FUNCTION_BLOCK T_MockStateModule IMPLEMENTS I_StateModule
VAR_INPUT
  _currentState : UINT;
END_VAR

{warning 'add property implementation'}
PROPERTY CurrentState : UINT
GET
CurrentState := _currentState;
END_GET
END_PROPERTY

END_FUNCTION_BLOCK

(* stored: Version 1.1.0.1, ProductVersion 3.1.4024.12
   POU T_MockStateModule: Id {494731a3-e8ea-4298-9b19-67e585bf4363}, SpecialFunc None
   Property CurrentState: Id {42c943d7-3807-4dad-aa79-0e2eaba5dc8a}
   Get Get: Id {55a7497a-587c-405e-812f-a54ec1698e9c} *)
